TYPE stPose3D EXTENDS stPose :
STRUCT
	z : LREAL;
	rx : LREAL;
	ry : LREAL;
	rz : LREAL;
END_STRUCT
END_TYPE

(* stored: Version 1.1.0.1, ProductVersion 3.1.4026.18
   DUT stPose3D: Id {b1b2c3d4-5555-5555-5555-555555555555} *)
